FUNCTION_BLOCK FILE_WRITER_11_CIRCULAR_MOVE (* Writes equation coeficients to a file (11 coef) for CIRCULAR_MOVE block *)
  (* Standard: 61499-2 *)
  (* Version 1.0, 02-05-12, GASR, Universidade do Estado de Santa Catarina *)
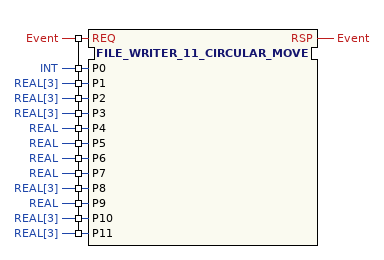
  EVENT_INPUT
    REQ WITH P0, P1, P2, P3, P4, P5, P6, P7, P8, P9, P10, P11; (* Request file storage *)
  END_EVENT
  EVENT_OUTPUT
    RSP; (* Finished operation *)
  END_EVENT
  VAR_INPUT
    P0 : INT; (* Process/equation id *)
    P1 : ARRAY [0..2] OF REAL; (* Coeficient 1 *)
    P2 : ARRAY [0..2] OF REAL; (* Coeficient 2 *)
    P3 : ARRAY [0..2] OF REAL; (* Coeficient 3 *)
    P4 : REAL; (* Coeficient 4 *)
    P5 : REAL; (* Coeficient 5 *)
    P6 : REAL; (* Coeficient 6 *)
    P7 : REAL; (* Coeficient 7 *)
    P8 : ARRAY [0..2] OF REAL; (* Coeficient 8 *)
    P9 : REAL; (* Coeficient 9 *)
    P10 : ARRAY [0..2] OF REAL; (* Coeficient 10 *)
    P11 : ARRAY [0..2] OF REAL; (* Coeficient 11 *)
  END_VAR
  SERVICE FILE_WRITER_11/MACHINE (* Coeficient file storage service *)
    SEQUENCE normal_establishment
      FILE_WRITER_11.REQ(P0,P1,P2,P3,P4,P5,P6,P7,P8,P9,P10,P11) -> MACHINE.write-file();
      MACHINE.response() -> FILE_WRITER_11.RSP();
    END_SEQUENCE
  END_SERVICE
END_FUNCTION_BLOCK
